Fanuc KAREL source: kc00028.KL

PROGRAM KC00028
%STACKSIZE=65535
%PRIORITY=65535
%NOLOCKGROUP
VAR
I : INTEGER
J : INTEGER
K : INTEGER
R : REAL
B : BOOLEAN
S : STRING[80]
T : STRING[80]
AI : ARRAY[8] OF INTEGER
JP : JOINTPOS9
P1 : POSITION
P2 : POSITION
P3 : POSITION
AR : ARRAY[9] OF REAL
-- UNRESOLVED DECLARATIONS (source type spelling not recovered)
-- P : TYPE_0x001F (type_u16=0x001F)
-- Q : TYPE_0x001F (type_u16=0x001F)
-- AB : ARRAY[244] OF TYPE_0x0018 (type_u16=0x2018)
-- C : TYPE_0x001C (type_u16=0x001C)
BEGIN
POS2JOINT(JP,P1,P2,P3,I,C,AR,JP,J)
END KC00028
